FUNCTION TryConvert_DATE_TO_SINT : BOOL
VAR_INPUT
	in : DATE;
	out : REFERENCE TO SINT;
END_VAR

IF in > SINT_TO_DATE(127) THEN
	RETURN;
END_IF

out := DATE_TO_SINT(in);
TryConvert_DATE_TO_SINT := TRUE;

END_FUNCTION

(* stored: Version 1.1.0.1, ProductVersion 3.1.4024.12
   POU TryConvert_DATE_TO_SINT: Id {59485a94-f235-4e24-91af-0d5aebccfba4}, SpecialFunc None *)
